Staubli VAL3: Key_ListBase.pgx

program Key_ListBase(bool& x_bRefresh, num& x_nKeyValue, num& x_nSelectItem)
begin
  x_bRefresh=true
  x_nKeyValue=getKey()
    switch x_nKeyValue
    //向上
    case 261
      x_nSelectItem=x_nSelectItem-1
    break
    //向下
    case 266
      x_nSelectItem=x_nSelectItem+1
    break

    default
      x_bRefresh=false
    break

    endSwitch

end
